(* Logix 5000 project; controller prova35v0 1756-L85E rev 35.11; software revision 35.00 *)

TASK MainTask (continuous, watchdog 500 ms) : MainProgram

MODULES
   Local : 1756-L85E (ICP 1, rev 35.11)
END_MODULES

VAR_GLOBAL   (* controller tags *)
   IoT_data : DINT;
END_VAR

PROGRAM MainProgram   (* main routine MainRoutine *)

ROUTINE MainRoutine   (* ladder *)
END_ROUTINE
END_PROGRAM
